{attribute addProperty BoxType "EPP2316-0003-0018"}
{attribute addProperty Id "DIG_InputsAT %I*DIG_Inputs_62B57CC87290DIG_Diag_InputsAT %I*DIG_Diag_Inputs_AC4A9AF06480DIG_Inputs_DeviceAT %I*DIG_Inputs_Device_D558E22E4050DIG_OutputsAT %Q*DIG_Outputs_33B763766480DIG_Outputs_DeviceAT %Q*DIG_Outputs_Device_735003021620WcStateAT %I*WcState_98A4DF7520.250InfoDataAT %I*InfoData_BC63D37F80100"}
{attribute addProperty CRC "532873803"}
{attribute addProperty SizeInBites "338"}
{attribute addProperty SizeInBytes "42.25"}
TYPE EPP2316_BCC80C64 :
STRUCT
	{attribute addProperty Name "DIG_Inputs"}
	DIG_Inputs : DIG_Inputs_62B57CC8;
	{attribute addProperty Name "DIG_Diag_Inputs"}
	DIG_Diag_Inputs : DIG_Diag_Inputs_AC4A9AF0;
	{attribute addProperty Name "DIG_Inputs_Device"}
	DIG_Inputs_Device : DIG_Inputs_Device_D558E22E;
	{attribute addProperty Name "DIG_Outputs"}
	DIG_Outputs : DIG_Outputs_33B76376;
	{attribute addProperty Name "DIG_Outputs_Device"}
	DIG_Outputs_Device : DIG_Outputs_Device_73500302;
	{attribute addProperty Name "WcState"}
	WcState : WcState_98A4DF75;
	{attribute addProperty Name "InfoData"}
	InfoData : InfoData_BC63D37F;
END_STRUCT
END_TYPE

(* stored: Version 1.2.0.0, ProductVersion 3.1.4024.9
   DUT EPP2316_BCC80C64: Id {2dcbfc1f-33a5-49f8-bfb0-50e259b8d307} *)
